// TIA Portal V20 export
DATA_BLOCK "ShiftmodelInterfaceHmi"   // DB103
TITLE = ShiftmodelTimes
AUTHOR : SICAR
FAMILY : Shiftmodel
VERSION : 1.0
// Global DB for HMI interface
// stored: InstanceOfName LSicar_typeShiftmodelHmi, InstanceOfType UDT
"LSicar_typeShiftmodelHmi"
   // VAR RETAIN
   //    shiftTimesListIndex : DInt;
   //    actualTimesDay : Array[0..7] of "LSicar_typeShiftmodTime1Day";
   //    actualSignalsDay : Array[0..7] of "LSicar_typeShiftmodSign1Day";
   //    summary : "LSicar_typeShiftmodSumHmi";
   //    actualDay : USInt;
   //    shiftTimesListOnOff : Bool := TRUE;   // Shift times OnOff
   //    setAdjTimes : Bool;
   //    hmiTimesValidFor : Array[0..3] of "LSicar_typeWeekdayBools";
   //    hmiTimes : Array[0..3] of "LSicar_typeShiftmodTime1Shift";   // Interface Local Times (Input on HMI)
   //    productionTimes : "LSicar_typeProdTimesHmi";
   // END_VAR
BEGIN
   hmiTimes[1].endCircuitTime := TOD#05:57:00;
   hmiTimes[2].endCircuitTime := TOD#13:57:00;
   hmiTimes[3].endCircuitTime := TOD#21:57:00;
   hmiTimes[1].start := TOD#06:00:00;
   hmiTimes[2].start := TOD#14:00:00;
   hmiTimes[3].start := TOD#22:00:00;
   hmiTimes[1].break[1].start := TOD#08:00:00;
   hmiTimes[1].break[2].start := TOD#10:00:00;
   hmiTimes[1].break[3].start := TOD#12:00:00;
   hmiTimes[1].break[4].start := TOD#00:00:00;
   hmiTimes[2].break[1].start := TOD#16:00:00;
   hmiTimes[2].break[2].start := TOD#18:00:00;
   hmiTimes[2].break[3].start := TOD#20:00:00;
   hmiTimes[2].break[4].start := TOD#00:00:00;
   hmiTimes[3].break[1].start := TOD#00:00:00;
   hmiTimes[3].break[2].start := TOD#02:00:00;
   hmiTimes[3].break[3].start := TOD#04:00:00;
   hmiTimes[3].break[4].start := TOD#00:00:00;
   hmiTimes[1].break[1].startCircuitTime := TOD#08:02:00;
   hmiTimes[1].break[2].startCircuitTime := TOD#00:00:00;
   hmiTimes[1].break[3].startCircuitTime := TOD#12:02:00;
   hmiTimes[1].break[4].startCircuitTime := TOD#00:00:00;
   hmiTimes[2].break[1].startCircuitTime := TOD#16:02:00;
   hmiTimes[2].break[2].startCircuitTime := TOD#00:00:00;
   hmiTimes[2].break[3].startCircuitTime := TOD#20:02:00;
   hmiTimes[2].break[4].startCircuitTime := TOD#00:00:00;
   hmiTimes[3].break[1].startCircuitTime := TOD#00:02:00;
   hmiTimes[3].break[2].startCircuitTime := TOD#00:00:00;
   hmiTimes[3].break[3].startCircuitTime := TOD#04:02:00;
   hmiTimes[3].break[4].startCircuitTime := TOD#00:00:00;
   hmiTimes[1].break[1].endCircuitTime := TOD#08:13:00;
   hmiTimes[1].break[2].endCircuitTime := TOD#00:00:00;
   hmiTimes[1].break[3].endCircuitTime := TOD#12:13:00;
   hmiTimes[1].break[4].endCircuitTime := TOD#00:00:00;
   hmiTimes[2].break[1].endCircuitTime := TOD#16:13:00;
   hmiTimes[2].break[2].endCircuitTime := TOD#00:00:00;
   hmiTimes[2].break[3].endCircuitTime := TOD#20:13:00;
   hmiTimes[2].break[4].endCircuitTime := TOD#00:00:00;
   hmiTimes[3].break[1].endCircuitTime := TOD#00:13:00;
   hmiTimes[3].break[2].endCircuitTime := TOD#00:00:00;
   hmiTimes[3].break[3].endCircuitTime := TOD#04:13:00;
   hmiTimes[3].break[4].endCircuitTime := TOD#00:00:00;
   hmiTimes[1].break[1].end := TOD#08:15:00;
   hmiTimes[1].break[2].end := TOD#10:10:00;
   hmiTimes[1].break[3].end := TOD#12:15:00;
   hmiTimes[1].break[4].end := TOD#00:00:00;
   hmiTimes[2].break[1].end := TOD#16:15:00;
   hmiTimes[2].break[2].end := TOD#18:10:00;
   hmiTimes[2].break[3].end := TOD#20:15:00;
   hmiTimes[2].break[4].end := TOD#00:00:00;
   hmiTimes[3].break[1].end := TOD#00:15:00;
   hmiTimes[3].break[2].end := TOD#02:10:00;
   hmiTimes[3].break[3].end := TOD#04:15:00;
   hmiTimes[3].break[4].end := TOD#00:00:00;
   hmiTimes[1].end := TOD#13:30:00;
   hmiTimes[2].end := TOD#21:30:00;
   hmiTimes[3].end := TOD#05:30:00;
   hmiTimes[1].startCircuitTime := TOD#13:33:00;
   hmiTimes[2].startCircuitTime := TOD#21:33:00;
   hmiTimes[3].startCircuitTime := TOD#05:33:00;
END_DATA_BLOCK
